// TIA Portal V19 export
TYPE "PPrf_A02_S1_PartsCutting"
// stored: Access Published
   STRUCT
      Rollformer { S7_SetPoint := 'True'} : "PPrf_Rollformer";
   END_STRUCT;
END_TYPE
